Staubli VAL3: F2_r2home.pgx

program F2_r2home()
begin
  //robot 2 move home position
  socket="(RBREDY)"
  watch(bRb2Ready,10)
  if bRb2Ready==true
    TcpStrRec:nFeedback=52
    //
    popUpMsg("Robot 2 is ready!")
  else
    //popUpMsg("Robot 2 is not ready!")
  endIf
end
